// TIA Portal V16 export
// export: Created 2021-09-01T08:19:45.3825186Z, ExportSetting WithDefaults, DisplayName Totally Integrated Automation Portal, DisplayVersion V16 Update 3, DisplayName TIA Portal Version Control Interface, DisplayVersion V16 Update 2, DisplayName TIA Portal Openness, DisplayVersion V16 Update 3, DisplayName TIA Portal Teamcenter Gateway, DisplayVersion V16, DisplayName STEP 7 Professional, DisplayVersion V16 Update 3, DisplayName STEP 7 Safety, DisplayVersion V16, DisplayName WinCC Advanced, DisplayVersion V16 Update 3
DATA_BLOCK "Sequencer_DB"   // DB17
VERSION : 0.1
// stored: AutoNumber true, DBAccessibleFromOPCUA true, InstanceOfName Sequencer, InstanceOfType FB
"Sequencer"
   // VAR_OUTPUT
   //    Dev1 : Bool;
   //    Dev2 : Bool;
   //    Dev3 : Bool;
   //    Dev4 : Bool;
   //    Dev5 : Bool;
   //    Dev6 : Bool;
   //    Dev7 : Bool;
   //    Dev8 : Bool;
   //    Dev9 : Bool;
   //    Dev10 : Bool;
   //    Dev11 : Bool;
   //    Dev12 : Bool;
   //    Dev13 : Bool;
   //    Dev14 : Bool;
   //    Dev15 : Bool;
   //    Dev16 : Bool;
   //    CurTime : Time;
   // END_VAR
   // VAR
   //    Enable : Bool;
   //    Hold : Bool;
   //    Seq { S7_SetPoint := 'True'} : "Sequence";
   //    RstStep { S7_SetPoint := 'True'} : Bool;
   //    "Step" : Int;
   //    Timer_IN { ExternalAccessible := 'False'; ExternalVisible := 'False'; ExternalWritable := 'False'} : Bool;
   //    Done : Bool;
   //    tmr { S7_SetPoint := 'True'} : "tmr200ms";
   // END_VAR
BEGIN
END_DATA_BLOCK
